PROGRAM pouS1Warnings
VAR
	
idbMsgWarn: FB_CheckMessageBounds;
END_VAR

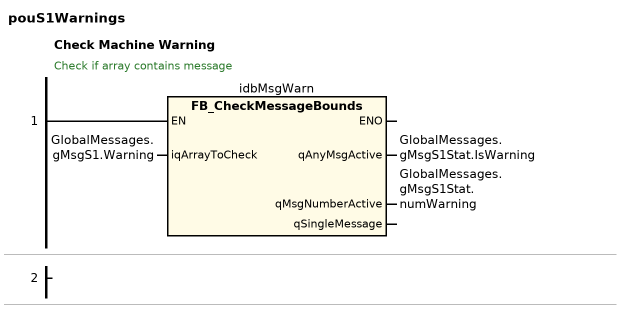
// NETWORK 1: Check Machine Warning
// Check if array contains message
idbMsgWarn(
    iqArrayToCheck := GlobalMessages.gMsgS1.Warning,
    qAnyMsgActive => GlobalMessages.gMsgS1Stat.IsWarning,
    qMsgNumberActive => GlobalMessages.gMsgS1Stat.numWarning); // FB_CheckMessageBounds

// NETWORK 2

END_PROGRAM

(* stored: Version 1.1.0.1, ProductVersion 3.1.4024.12
   POU pouS1Warnings: Id {65a0745a-e675-400f-ad40-91f4efb6ca28}, SpecialFunc None *)
